FUNCTION_BLOCK F_CEIL (* returns the smallest possible integer which is greater or equal to X *)
  (* Standard: OSCAT; Classification: Math *)
  (* Version 0.0, 2011-07-21, 4DIAC-IDE, 4DIAC-Consortium *)
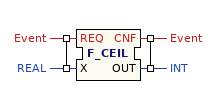
  EVENT_INPUT
    REQ WITH X; (* Service Request *)
  END_EVENT
  EVENT_OUTPUT
    CNF WITH OUT; (* Confirmation of Requested Service *)
  END_EVENT
  VAR_INPUT
    X : REAL; (* Input *)
  END_VAR
  VAR_OUTPUT
    OUT : INT; (* Outcome *)
  END_VAR
END_FUNCTION_BLOCK
